// TIA Portal V21 export
VAR_GLOBAL   // PLC tag table "Process_Data"
   IB_Byte0 AT %IB400 : Byte;
   IB_Byte1 AT %IB401 : Byte;
   OB_Byte0 AT %QB400 : Byte;
   OB_Byte1 AT %QB401 : Byte;
   OB_Byte2 AT %QB402 : Byte;
   OB_Byte3 AT %QB403 : Byte;
   OB_Byte4 AT %QB404 : Byte;
   OB_Byte5 AT %QB405 : Byte;
   OB_Byte6 AT %QB406 : Byte;
   OB_Byte7 AT %QB407 : Byte;
   OB_Byte8 AT %QB408 : Byte;
   OB_Byte9 AT %QB409 : Byte;
   OB_Byte10 AT %QB410 : Byte;
   IB_Byte2 AT %IB402 : Byte;
   IB_Byte3 AT %IB403 : Byte;
   OB_Byte11 AT %QB411 : Byte;
END_VAR
